// Mitsubishi GX Works2 project: 240430_timechart04_직렬회로gxw   PLC: Q03UDV

PROGRAM MAIN
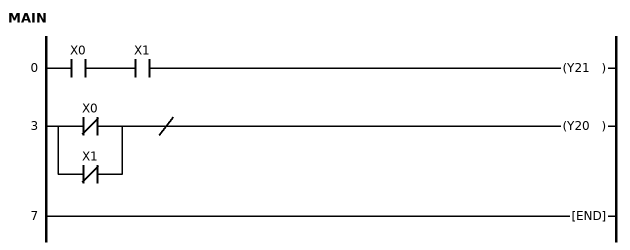
0     LD      X0
      AND     X1
      OUT     Y21
3     LDI     X0
      ORI     X1
      INV
      OUT     Y20
7     END
END_PROGRAM
